FUNCTION_BLOCK EquipmentModule EXTENDS FB_PackML_BaseModule IMPLEMENTS ITF_Observer
VAR
	NextState		: BOOL;
	AbortReq		: BOOL;
	
	
	//ITF_Observable
	OModule : REFERENCE TO MachineModule;

	//
	interlock : Interlock;
	reqDoStuff: BOOL;
	stuffDone: BOOL;
END_VAR

METHOD PUBLIC CyclicLogic
VAR
END_VAR
IF NOT _InitComplete THEN
	_InitComplete := Initialize();
	RETURN;
END_IF

//Check Interlock
IF reqDoStuff THEN
	reqDoStuff := FALSE;
	IF interlock.Unlocked THEN
		IF __ISVALIDREF(OModule) THEN
			OModule.Lock(THIS^); //Lock the interlock
		END_IF

		//OK to do stuff
	ELSE
		//Locked
		IF __ISVALIDREF(OModule) THEN
			TRACE(CONCAT(STR1 := 'Interlock set by: ', STR2 := TO_STRING(OModule.InterlockList)));
		END_IF
	END_IF
END_IF

//Release Interlock
IF stuffDone AND interlock.Locked THEN
	stuffDone := FALSE;
	IF __ISVALIDREF(OModule) THEN
		OModule.Unlock(THIS^);
	END_IF
END_IF

SUPER^.CyclicLogic();
END_METHOD

METHOD PROTECTED Initialize : BOOL
Initialize := TRUE;
END_METHOD

METHOD updateConnection
VAR_INPUT
	Module : REFERENCE TO MachineModule;
END_VAR
OModule REF= Module;
END_METHOD

METHOD updateLock
VAR_INPUT
	setLock : BOOL;
END_VAR
//Method called by observable to notify of lock status
IF setLock THEN
	interlock.Lock();
ELSE
	interlock.Unlock();
END_IF
END_METHOD

END_FUNCTION_BLOCK

(* stored: Version 1.1.0.1, ProductVersion 3.1.4024.12
   POU EquipmentModule: Id {f2e656c0-93da-44d4-9459-07fffe962a19}, SpecialFunc None
   Method CyclicLogic: Id {a78de6c5-4a2b-4916-a597-ad8bb018c6f0}
   Method Initialize: Id {00c6170c-354e-46b1-b773-30d5828110ec}
   Method updateConnection: Id {2e52bece-f250-4467-b7ad-cd7fd7b9e6c1}
   Method updateLock: Id {e40c8d18-8c90-46d4-8156-7cc4a664175f} *)
